FUNCTION FC_Instances : BOOL
VAR_INPUT
END_VAR
VAR
END_VAR

// Befehlsverarbeitung
Sequencer(
	sPath			:= GVL_ProgramSequencer.Sequencer.sPath,
	bPelletsEmpty	:= GVL_HardwareExtruder.I_PelletsEmpty,
	bReady 			=> GVL_ProgramSequencer.Sequencer.bReady,
	bPrinting 		=> GVL_ProgramSequencer.Sequencer.bPrinting,
	bFinished		=> GVL_ProgramSequencer.Sequencer.bFinished,
	bError        	=> GVL_ProgramSequencer.Sequencer.bError,
	nErrorID      	=> GVL_ProgramSequencer.Sequencer.nErrorID,
	sErrorMsg 		=> GVL_ProgramSequencer.Sequencer.sErrorMsg,
	bHeatersEnabled	:= GVL_ProgramSequencer.Sequencer.bHeatersEnabled,
	bPrintBedClear	:= GVL_ProgramSequencer.Sequencer.bPrintBedClear,
	bChangeMaterial	:= GVL_ProgramSequencer.Sequencer.bChangeMaterial,
	bChangeMaterialFinished := GVL_ProgramSequencer.Sequencer.bChangeMaterialFinished,
	bLoadFile		:= GVL_ProgramSequencer.Sequencer.bLoadFile,
	bCloseFile		:= GVL_ProgramSequencer.Sequencer.bCloseFile,
	bStart 			:= GVL_ProgramSequencer.Sequencer.bStart,
	bAbort 			:= GVL_ProgramSequencer.Sequencer.bAbort,
	bPause          := GVL_ProgramSequencer.Sequencer.bPause,
	bResume         := GVL_ProgramSequencer.Sequencer.bResume,
	bErrorReset 	:= GVL_ProgramSequencer.Sequencer.bErrorReset);

// Druckbett
PrintingBed(
	bErrorReset		:= GVL_PrintingBed.PrintingBed.bErrorReset,
	bError			=> GVL_PrintingBed.PrintingBed.bError,
	nErrorID		=> GVL_PrintingBed.PrintingBed.nErrorID,
	sErrorMsg		=> GVL_PrintingBed.PrintingBed.sErrorMsg);

// Extruder	
ExtruderControl(
	bErrorReset		:= GVL_Extruder.Extruder.bErrorReset,
	bHeatersEnabled := GVL_ProgramSequencer.Sequencer.bHeatersEnabled,
	bReady			=> GVL_Extruder.Extruder.bReady,
	bExtruding		=> GVL_Extruder.Extruder.bExtruding,
	bHeatingActiv	=> GVL_Extruder.Extruder.bHeatingActiv,
	bError			=> GVL_Extruder.Extruder.bError,
	nErrorID      	=> GVL_Extruder.Extruder.nErrorID,
    sErrorMsg 		=> GVL_Extruder.Extruder.sErrorMsg,
	bStartHeater	:= GVL_Extruder.Extruder.bStartHeater,
	bStopHeater		:= GVL_Extruder.Extruder.bStopHeater,
	bStart			:= GVL_Extruder.Extruder.bStart,
	bStop			:= GVL_Extruder.Extruder.bStop);	

// Heizelemente
HeaterTop(
	bEnable			:= GVL_Extruder.HeaterTop.bEnabled,
    fSetTemp		:= GVL_ParameterExtruder.aMaterialSettings[GVL_ParameterExtruder.nMaterial].fTempTop,
	fPID_Output     => GVL_Extruder.HeaterTop.fPID_Output,
	bAtTemp         => GVL_Extruder.HeaterTop.bAtTemp,
    bErrorReset		:= GVL_Extruder.HeaterTop.bErrorReset,
    bError        	=> GVL_Extruder.HeaterTop.bError,
    nErrorID      	=> GVL_Extruder.HeaterTop.nErrorID,
    sErrorMsg 		=> GVL_Extruder.HeaterTop.sErrorMsg,
	fWarmupKp       := GVL_ParameterExtruder.WarmupHeaterTop.fKp,
	fWarmupKi       := GVL_ParameterExtruder.WarmupHeaterTop.fKi,
	fWarmupKd       := GVL_ParameterExtruder.WarmupHeaterTop.fKd,
	fWarmupFilterN 	:= GVL_ParameterExtruder.WarmupHeaterTop.fFilterN,
	bPrinting		:= GVL_Extruder.Extruder.bExtruding,
	fPrintingKp     := GVL_ParameterExtruder.PrintingHeaterTop.fKp,
	fPrintingKi     := GVL_ParameterExtruder.PrintingHeaterTop.fKi,
	fPrintingKd     := GVL_ParameterExtruder.PrintingHeaterTop.fKd,
	fPrintingFilterN:= GVL_ParameterExtruder.PrintingHeaterTop.fFilterN,
	tRampTime		:= GVL_ParameterExtruder.tRampTime,
	nPIDCycleFactor	:= GVL_ParameterExtruder.nPIDCycleFactor,
	tPWM_Period     := GVL_ParameterExtruder.tPWM_Period,
	fAtTempTolerance:= GVL_ParameterExtruder.fAtTempTolerance,
	nTempRaw		:= GVL_HardwareExtruder.I_TempRaw_Top,
	fActualTemp		=> GVL_Extruder.HeaterTop.fActualTemp,
	bSSR_Out		=> GVL_HardwareExtruder.Q_SSR_Top);

HeaterMiddle(
	bEnable			:= GVL_Extruder.HeaterMiddle.bEnabled,
    fSetTemp		:= GVL_ParameterExtruder.aMaterialSettings[GVL_ParameterExtruder.nMaterial].fTempMiddle,
	fPID_Output     => GVL_Extruder.HeaterMiddle.fPID_Output,
	bAtTemp         => GVL_Extruder.HeaterMiddle.bAtTemp,
    bErrorReset		:= GVL_Extruder.HeaterMiddle.bErrorReset,
    bError        	=> GVL_Extruder.HeaterMiddle.bError,
    nErrorID      	=> GVL_Extruder.HeaterMiddle.nErrorID,
    sErrorMsg 		=> GVL_Extruder.HeaterMiddle.sErrorMsg,
	fWarmupKp       := GVL_ParameterExtruder.WarmupHeaterMiddle.fKp,
	fWarmupKi       := GVL_ParameterExtruder.WarmupHeaterMiddle.fKi,
	fWarmupKd       := GVL_ParameterExtruder.WarmupHeaterMiddle.fKd,
	fWarmupFilterN 	:= GVL_ParameterExtruder.WarmupHeaterMiddle.fFilterN,
	bPrinting		:= GVL_Extruder.Extruder.bExtruding,
	fPrintingKp     := GVL_ParameterExtruder.PrintingHeaterMiddle.fKp,
	fPrintingKi     := GVL_ParameterExtruder.PrintingHeaterMiddle.fKi,
	fPrintingKd     := GVL_ParameterExtruder.PrintingHeaterMiddle.fKd,
	fPrintingFilterN:= GVL_ParameterExtruder.PrintingHeaterMiddle.fFilterN,
	tRampTime		:= GVL_ParameterExtruder.tRampTime,
	nPIDCycleFactor	:= GVL_ParameterExtruder.nPIDCycleFactor,  
	tPWM_Period     := GVL_ParameterExtruder.tPWM_Period,      
	fAtTempTolerance:= GVL_ParameterExtruder.fAtTempTolerance,
	nTempRaw		:= GVL_HardwareExtruder.I_TempRaw_Middle,
	fActualTemp		=> GVL_Extruder.HeaterMiddle.fActualTemp,
	bSSR_Out		=> GVL_HardwareExtruder.Q_SSR_Middle);
		
HeaterNozzle(
	bEnable			:= GVL_Extruder.HeaterNozzle.bEnabled,
    fSetTemp		:= GVL_ParameterExtruder.aMaterialSettings[GVL_ParameterExtruder.nMaterial].fTempNozzle,
	fPID_Output     => GVL_Extruder.HeaterNozzle.fPID_Output,
	bAtTemp         => GVL_Extruder.HeaterNozzle.bAtTemp,
    bErrorReset		:= GVL_Extruder.HeaterNozzle.bErrorReset,
    bError        	=> GVL_Extruder.HeaterNozzle.bError,
    nErrorID      	=> GVL_Extruder.HeaterNozzle.nErrorID,
    sErrorMsg 		=> GVL_Extruder.HeaterNozzle.sErrorMsg,
	fWarmupKp       := GVL_ParameterExtruder.WarmupHeaterNozzle.fKp,
	fWarmupKi       := GVL_ParameterExtruder.WarmupHeaterNozzle.fKi,
	fWarmupKd       := GVL_ParameterExtruder.WarmupHeaterNozzle.fKd,
	fWarmupFilterN 	:= GVL_ParameterExtruder.WarmupHeaterNozzle.fFilterN,
	bPrinting		:= GVL_Extruder.Extruder.bExtruding,
	fPrintingKp     := GVL_ParameterExtruder.PrintingHeaterNozzle.fKp,
	fPrintingKi     := GVL_ParameterExtruder.PrintingHeaterNozzle.fKi,
	fPrintingKd     := GVL_ParameterExtruder.PrintingHeaterNozzle.fKd,
	fPrintingFilterN:= GVL_ParameterExtruder.PrintingHeaterNozzle.fFilterN,
	tRampTime		:= GVL_ParameterExtruder.tRampTime,
	nPIDCycleFactor	:= GVL_ParameterExtruder.nPIDCycleFactor,  
	tPWM_Period     := GVL_ParameterExtruder.tPWM_Period,      
	fAtTempTolerance:= GVL_ParameterExtruder.fAtTempTolerance,
	nTempRaw		:= GVL_HardwareExtruder.I_TempRaw_Nozzle,
	fActualTemp		=> GVL_Extruder.HeaterNozzle.fActualTemp,
	bSSR_Out		=> GVL_HardwareExtruder.Q_SSR_Nozzle);

//Motor
ExtruderMotor(
	bEnable			:= GVL_Extruder.ExtruderMotor.bEnable,
	bErrorReset		:= GVL_Extruder.ExtruderMotor.bErrorReset,
	fSetRPM			:= GVL_ParameterExtruder.fMotorRPM,
	bError_Stepper	:= GVL_HardwareExtruder.I_Stepper.bError,
	bStepper_STALL	:= GVL_HardwareExtruder.I_Stepper.bStallguardActive,
	bRunning		=> GVL_Extruder.ExtruderMotor.bRunning,
	bError			=> GVL_Extruder.ExtruderMotor.bError,
	nErrorID		=> GVL_Extruder.ExtruderMotor.nErrorID,
	sErrorMsg		=> GVL_Extruder.ExtruderMotor.sErrorMsg,
	nPTO_FreqValue	=> GVL_HardwareExtruder.Q_Stepper.nFrequencyValue,
	n_Direction		=> GVL_HardwareExtruder.Q_Stepper.nDirection,
	n_Enable		=> GVL_HardwareExtruder.Q_Stepper.nEnable);

END_FUNCTION

(* stored: Version 1.1.0.1
   POU FC_Instances: Id {24fadc25-913a-4aa8-9ee9-bd4c3f715ed4}, SpecialFunc None *)
